// TIA Portal V20 export
TYPE "LKinCtrl_typeConfigurationAxis"
// stored: Access Published
   STRUCT
      "name" { ExternalAccessible := 'False'; ExternalVisible := 'False'; ExternalWritable := 'False'; S7_SetPoint := 'True'} : WString["LKINCTRL_LENGTH_OF_TO_NAME"];   // Axis name shown on HMI
      used { ExternalAccessible := 'False'; ExternalVisible := 'False'; ExternalWritable := 'False'; S7_SetPoint := 'True'} : Bool := FALSE;   // TRUE: axis is activated for HMI use, FALSE: axis is deactivated for HMI use / TRUE: Axis is used (only relevant for additional axes, kinematic axes are always used)
      withBrake { ExternalAccessible := 'False'; ExternalVisible := 'False'; ExternalWritable := 'False'; S7_SetPoint := 'True'} : Bool := FALSE;   // TRUE: Axis has a motor holding brake
      homePosition { ExternalAccessible := 'False'; ExternalVisible := 'False'; ExternalWritable := 'False'; S7_SetPoint := 'True'} : LReal := 0.0;   // Defines the default homing position
      coupling { ExternalAccessible := 'False'; ExternalVisible := 'False'; ExternalWritable := 'False'; S7_SetPoint := 'True'} : Bool := FALSE;   // TRUE: Coupling present
      jog { ExternalAccessible := 'False'; ExternalVisible := 'False'; ExternalWritable := 'False'; S7_SetPoint := 'True'} : "LKinCtrl_typeJogConfiguration";
   END_STRUCT;
   // jog.accelerationTime := 0.2;
   // jog.maxVelocityManual := 10.0;
   // jog.maxVelocityTestRun := 10.0;
   // jog.presetIncrementCoarse := 5.0;
   // jog.presetIncrementFine := 1.0;
   // jog.presetIncrementPrecise := 0.5;
END_TYPE
